{attribute wpf [Container(Layout.Wrap)]}
{attribute wpf [Group(Layout.GroupBox)]}
{attribute addProperty Name ""}
TYPE stContinuousValueLimits :
STRUCT	
	{attribute addProperty Name "<#Min#>"}
	Minimum : REAL;		
	{attribute addProperty Name "<#Acquired#>"}
	{attribute wpf [RenderIgnore("Control", "ShadowControl")]} // Prevents rednering this memember when 'PresentationType' is set to 'Control' or 'ShadowControl'.
	Acquired : REAL;	
	{attribute addProperty Name "<#Max#>"}
	Maximum : REAL;
END_STRUCT
END_TYPE

(* stored: Version 1.1.0.1, ProductVersion 3.1.4024.3
   DUT stContinuousValueLimits: Id {46de2d8f-e96c-49d9-a008-9e1b5b9871a5} *)
